(* CODESYS project Enums.export

Project tree, tasks and I/O mapping:
  Enums/
    data type DepositeProcessStage
    data type ERROR
    data type InficonMethodStage
    data type InficonMethodStatus
    data type InficonStage
    data type IPS_CONTROL_STAGE
    data type IPS_STATUS
    data type OWEN_TYPE
    data type PRESSURE_UNIT
    data type VACUUM_CAMERA_PROCESS_STAGE
    data type VACUUM_CAMERA_STATE
    TRM151/
      data type TRMAutomationCorrectionFreeEnds
      data type TRMInputNumberTrancitionValue
      data type TRMInputSensoreType
      data type TRMmanualChangeValue
      data type TRMNextStepTransactionLogic
      data type TRMObjectState
      data type TRMProgramPermit
      data type TRMRegulationMode
      data type TRMSetpointType
      data type TRMStartProgramSource
      data type TRMStartSignal
      data type TRMStepType
      data type TRMTimeFormat
      data type TRMTransactionConditionValue
      data type TRM_POOLING_STAGE
*)

// Enums/DepositeProcessStage
{attribute 'qualified_only'}
{attribute 'strict'}

TYPE DepositeProcessStage :
(
	WAIT_COMMAND 			:=0,  //Ожидание команды на старт
	INIT_DATA				:=10, //Инициализация уставок
	START_HEATER			:=11, //Включение источчника питания
	PREDEPOSITE_HEATING		:=15, //Этап нагрева по времени
	QARTZ_OPEN				:=20, //Открытие клапана кварцевого датчика
	QUARTZ_OPENED_DELAY		:=21, //Ожидание при открытом кварцевом датчике
	SOURCE_SHUTTER_OPEN		:=25, //Открытие залсонку источника напыления
	QARTZ_SENSORE_HEATING	:=30, //Прогрев кварцевого датчика для стабилизации показаний
	LIMIT_SPEED_DEPOSITE_1	:=35, //Напыление с заданной скоростью
	LIMIT_SPEED_DEPOSITE_2	:=36, //Наплыение с заданной скоростью
	STOP_DEPOSITE			:=40, //Остановка напыления
	ERROR					:=100 //Ошибка 
);
END_TYPE

// Enums/ERROR
{attribute 'qualified_only'}
//{attribute 'conditionalshow'}
//{attribute 'conditionalshow' := 'SomeText'}
//{attribute 'hide'}
TYPE ERROR : (NO_ERROR, TIME_OUT); END_TYPE

// Enums/InficonMethodStage
{attribute 'qualified_only'}
{attribute 'strict'}
TYPE InficonMethodStage :
(
	WAIT := 0,
	ADD_COMMAND:=1,
	ADD_LENGTH_TO_SENDBUFFER:=61,
	CALC_CRC:=70,
	ADD_CRC:=80,
	ADD_DATA_TO_SENDBUFFER:=90,
	EDGE_MESSAGECOMPLETE_FLAG:=91,
	WAIT_RESPONCE:=110,
	PARSE_RESPONCE:=120,
	CHECK_RESPONCE_STATUS:=121,
	COMPLETE:=130,
	ERROR:=140
);
END_TYPE

// Enums/InficonMethodStatus
{attribute 'qualified_only'}
{attribute 'strict'}
TYPE InficonMethodStatus :
(
	IDLE := 0,
	BUSY:=1,
	COMPLETE:=100,
	ERROR:=255
);
END_TYPE

// Enums/InficonStage
{attribute 'qualified_only'}
{attribute 'strict'}
TYPE InficonStage :
(
	WAIT := 0,
	STATUS_SENSORE:=10,
	GET_MATERIAL_FILTRED_RATE:=20,
	REMOTE_GENERAL_ACTION:=30,
	ERROR:=100
);
END_TYPE

// Enums/IPS_CONTROL_STAGE
{attribute 'qualified_only'}
{attribute 'strict'}
TYPE IPS_CONTROL_STAGE :
(
	WAIT := 0,
	START_PERMIT:=10,
	WAIT_PERMIT_ANSWER:=11,
	START:=20,
	WAIT_START_RESPONCE:=21,
	STOP:=30,
	WAIT_STOP_RESPONCE:=31,
	ERROR_RESET:=40,
	WAIT_ERROR_RESET_RESPONCE:=41,
	ERROR:=100
);
END_TYPE

// Enums/IPS_STATUS
{attribute 'qualified_only'}
{attribute 'strict'}
{attribute 'to_string'}
TYPE IPS_STATUS :
(
	PROCESS_RESET := 				769,	//Прошла инициализация устрйоства после включения питания
	START_PERMIT:=					10101,	//Разрешение выполнения ккоманды "Старт" выполнено без ошибок
	START_NO_ERROR:=				10001,	//Команда "старт" с  выполнена без ошибок
	START_KEYBORD_NO_ERROR:=		10201,	//Команда "старт" с клавитауры ввыполнена без ошибок
	START_CONTACT_NO_ERROR:=		10301, 	//Команда "Старт" с внешнего контакта выполнена без ошибок
	RUN_STEP_1:=					30101, 	//Выполняется команда "Старт" шаг 1
	RUN_STEP_2:=					30201,	//Выполняется команда "Старт" шаг 2
	RUN_STEP_3:=					30301,	//Выполняется команда "Старт" шаг 3
	RUN_STEP_4:=					30401,	//Выполняется команда "Старт" шаг 4
	RUN_STEP_5:=					30501,  //Выполняется команда "Старт" шаг 5
	RUN_STEP_6:=					30601,	//Выполняется команда "Старт" шаг 6
	RUN_STEP_7:=					30701,	//Выполняется команда "Старт" шаг 7
	RUN_STEP_7_1:=					30711, 	//Выполняется команда "Старт" шаг 7.1
	RUN_STEP_7_2:=					30721,	//Выполняется команда "Старт" шаг 7.2
	RUN_STEP_7_3:=					30731,	//Выполняется команда "Старт" шаг 7.3
	RUN_STEP_8:=					30801,	//Выполняется команда "Старт" шаг 8
	RUN_STEP_9:=					30901,	//Выполняется команда "Старт" шаг 9
	ERR_START_PERMIT:=				40101,	//Ошибка выполнения команда "Старт", нет разрешения старта
	ERR_START_ALARM:=				40201,	//Ошибка выполнения команды "Старт", активен сигнал авария
	ERR_START_POWER_SUPPLY:=		40301,	//Ошибка выполнения команды "Старт", напряжение истоника питная собственных нужд ниже нормы
	ERR_START_HIGHT_TEMPERATURE:=	40401,	//Ошибка выполнения команды "Старт" высокая температура воздуха
	ERR_START_HIGHT_TEMPERATURE_1:=	40501,	//Ошибка выполнения команды "Старт" высокая температура узлов устройства
	ERR_START_HIGHT_TEMPERATURE_2:= 40601,
	ERR_START_HIGHT_TEMPERATURE_3:= 40701,
	ERR_START_HIGHT_TEMPERATURE_4:= 41101,
	ERR_START_BLOCK_CONTACT:=		41001,	//Ошибка выполнения команды "Старт" контакт блокировки отключен
	ERR_START_ALREADY:=				41201,	//Ошибка выполнения команды "Старт" блок уже включен
	ERR_START_FILAMENT_CUT:=		41301,	//ошибка выполнения команды "Старт", обрыв нити накала
	ERR_START_GROUND_CUT:=			41501,	//Ошибка выполнения команды "Старт", обрыв заземления нагрузки
	ERR_START_DISPLAY_DISCONNECT:=	41601, 	//Ошибка выполнения команды "Старт", нет связи с дисплеем блока
	ERR_START_CONVERTER_MISSING:=	41701,	//Ошибка выполнения команды "Старт", нет подключенных преобразователей
	ERR_START_RMS_HOT:=				41801,	//Ошибка выполнения команды "Старт", датчик RMS горячий
	ERR_START_INTERNAL_CONNECT_1:=	41901,	//Ошибка выполнения команды "Старт", проблема со связью между узлами внутри блока
	ERR_START_INTERNAL_CONNECT_2:=	42001,
	ERR_START_INTERNAL_CONNECT_3:=	42101,
	ERR_START_STOP_DELAY:=			42201,	//Ошибка выполнения команды "Старт", пауза после выключения меньше 3 секунд
	ERR_START_RUN_CONVERTER_ERR:=	42301,	//Ошибка выполнения команды "Старт", проблемы с пуском преобразователя
	ERR_START_ADC_DISCONNECT:=		42601,	//Ошибка выполнения команды "Старт", нет связи с АЦП контроля выходного напрядения устройства
	STOP_NO_ERROR:=					10002,	//Команда "Стоп" выполнена
	STOP_KEYBORD_NO_ERROR:=			10102,	//Команда "Стоп" выполнена по нажатию кнопки "Стоп"
	STOP_CONTACT_NO_ERROR:=			10202,	//Команда "Стоп" выполнена по вненему контакту
	STOP_AFTER_SMOOTH_SHUTDOWN_FILAMENT:=	10501, //Команда "Стоп" выполнена после плавного отключения накала
	STOP_ANOD_CHANELL:=				10602,	//Команда "Стоп" выполнена для канала анода
	EMG_STOP_ALARM:=				40202,	//Аварийный "Стоп по сигналу "Авария"
	EMG_STOP_POWER_SUPPLY:=			40302,	//Аварийный "Стоп", напряжение источника питания собственных нужд ниже нормы
	EMG_STOP_HOT_AIR:=				40402,	//Авариынй "Стоп", горячий воздух
	EMG_STOP_OVERHEAT_1:=			40502,	//Аварийный "Стоп", перегрев узлоа
	EMG_STOP_OVERHEAT_2:=			40602,
	EMG_STOP_OVERHEAT_3:=			40702,
	EMG_STOP_OVERHEAT_4:=			41102,
	EMG_STOP_WATCHDOG:=				40802,	//Аварийный "Стоп" сработал сторожевой таймер
	EMG_STOP_INTERLOCK:=			41002,	//Аварийный "Стоп", сработал внешний блокировочный контакт
	EMG_STOP_FILAMENT_ALARM:=		41302,	//Аварийный "Стоп", авария накала
	EMG_STOP_INTERNAL_SYNC_MISSING:=41402,	//Аварийный "Стоп", потеря внетренней синхронизации между узлами устройства
	EMG_STOP_GROUND_CUT:=			41502,	//Аварийный "Стоп", обрыв заземления нагрузки
	EMG_STOP_INTERNAL_CONNECT_1:=	41602,	//аварийный "Стоп", ошибка связи между узлами устройства
	EMG_STOP_INTERNAL_CONNECT_2:=	41902,
	EMG_STOP_INTERNAL_CONNECT_3:=	42002,
	EMG_STOP_INTERNAL_CONNECT_4:=	42102,
	EMG_STOP_RMS_OVERLOAD:=			41802,	//Аварийный "Стоп", большой ток RMS
	EMG_STOP_CONVERTER_EMG_RELOAD:=	42202,	//Аварийный "Стоп", аварийный перезапуцск преобразователя
	EMG_STOP_LOW_VOLTAGE:=			42302,	//Аварийный "Стоп", напряжение нагрузки ниже нормы
	EMG_STOP_ADC_DISCONNECT:=		42602, 	//Аварийный "Стоп", нет связи с АЦП контроля выходного напряжения устройства
	RESET_ERROR_DONE:=				10003, 	//Команда "Сброс ошибок" выполнена
	RESET_ERROR_AFTER_STOP:=		10103, 	//Команда "Сброс ошибок" выполнена по нажатию кнопки "Стоп"
	RESET_ERROR_FAIl:=				40003	//Команда "Сброс ошибок" не выполнена, устройство в режиме "Старт"
	
);
END_TYPE

// Enums/OWEN_TYPE
{attribute 'qualified_only'}
{attribute 'strict'}
TYPE OWEN_TYPE :
(
	INTEGER 	:= 0,
	FLOAT		:=1,
	OTHER		:=2
);
END_TYPE

// Enums/PRESSURE_UNIT
{attribute 'qualified_only'}
{attribute 'strict'}
TYPE PRESSURE_UNIT :
(
	mBar := 0,
	Pascal:=1,
	Torr:=2
);
END_TYPE

// Enums/VACUUM_CAMERA_PROCESS_STAGE
{attribute 'qualified_only'}
{attribute 'strict'}
TYPE VACUUM_CAMERA_PROCESS_STAGE :
(
	WAIT := 0, //Ожидание
	START_VACUUM_PROCESS:=10,//Старт процессса откачки вакуумной камеры
	START_VACUUM_PROCESS_CHECK_FVP_SELECT:=11,//Проверка ФВП на флаг работоспособности
	START_VACUUM_PROCESS_CHECKING_FVP:=12,//Проверка ФВН на рпботоспособнтсть
	START_VACUUM_PROCESS_FORVACUUMING_PROCESS:=13,//Процесс форвакуумной откачка
	START_VACUUM_PROCESS_TMP_FORVACUUMING_PROCESS:=14,//Процесс откачки через форвакуумный насосо и ТМН
	START_VACUUM_PROCESS_TMP_START:=15,//Запуск ТМН
	START_VACUUM_PROCESS_COMPLETE_WAIT:=16,//Ожидание завершения процессаы
	START_REVACUUM_PROCESS:=20,//Старт процесса повтороной откачки вакуумнйо камеры
	
	
	START_DEVACUUM_PROCESS:=30,//Старт процесса напуска атмосферы в вакуумную камеру
	START_DEVACUUM_STOP_TMP:=31,//Старт полного цикла остановки
	START_DEVACUUM_STOP_FVP:=32,
	START_DEVACUUM_OPEN_CAM:=33,

	
	
	
	
	STOP_VACUUM_PROCESS:=40,//остановка работы вакуумной камеры
	STOP_ANY_PROCESS:=50, //Стадия остановки любого процесса
	ERROR:=1000//Ошибка в работе алгоритма
);
END_TYPE

// Enums/VACUUM_CAMERA_STATE
{attribute 'qualified_only'}
{attribute 'strict'}
TYPE VACUUM_CAMERA_STATE :
(
	CAMERA_NOT_VACUUM := 0,	//Камера находится не под вакуумом
	CAMERA_VACUUM:=10 		//Камера находится по двакуумом
	
);
END_TYPE

// Enums/TRM151/TRMAutomationCorrectionFreeEnds
{attribute 'qualified_only'}
{attribute 'strict'}
TYPE TRMAutomationCorrectionFreeEnds :
(
	OFF := 1,
	ON	:=2
);
END_TYPE

// Enums/TRM151/TRMInputNumberTrancitionValue
{attribute 'qualified_only'}
{attribute 'strict'}
(*
Номер входа, величина с которого должна достичь значение уставки
*)
TYPE TRMInputNumberTrancitionValue :
(
	OFF := 0,
	Input_1:=1,
	Input_2:=2
);
END_TYPE

// Enums/TRM151/TRMInputSensoreType
{attribute 'qualified_only'}
{attribute 'strict'}
TYPE TRMInputSensoreType :
(
	DISABLE := 0,
	TSM100M :=1,
	TSM50M:=2,
	TSP100P_1_385:=3,
	TSP100P_1_391:=4,
	THK_L:=5,
	THA_K:=6,
	Sensore50vM:=7,
	TSP50_1_385:=8,
	TSP50_1_391:=9,
	Sensore_4_20ma:=11,
	Sensore_0_20ma:=12,
	Sensore_0_5ma:=13,
	Sensore_0_1V:=14,
	TPR_B:=17,
	TPP_S:=18,
	TPP_R:=19,
	TNN_N:=20,
	TJK_J:=21,
	TVR_A_1:=22,
	TVR_A_2:=23,
	TVR_A_3:=24,
	TMK_T:=25
	
);
END_TYPE

// Enums/TRM151/TRMmanualChangeValue
{attribute 'qualified_only'}
{attribute 'strict'}
TYPE TRMmanualChangeValue :
(
	Enable := 0,
	Disable:=1
);
END_TYPE

// Enums/TRM151/TRMNextStepTransactionLogic
{attribute 'qualified_only'}
{attribute 'strict'}
(*Логика перехода на следующий шаг*)
TYPE TRMNextStepTransactionLogic :
(
	GetLimitValue := 1, //По достижению порогового ззначения
	GetTime:=2,			//по времения
	GetLimitValueAndtime:=3,//По достижению порогового значени и времени
	GetLimitValueOrtime:=4
);
END_TYPE

// Enums/TRM151/TRMObjectState
{attribute 'qualified_only'}
{attribute 'strict'}
TYPE TRMObjectState :
(
	Stop := 0,								//Останов
	Work:=1,								//Работа
	WaitWorkCondition:=2,					//Ожидание условий запуска
	Pause:=3,								//пауза
	WaitWorkConditionAfterPowerFailure:=4,	//Ожидание условй запуска после пропадания питания
	GraphicSetMode:=5,						//Режим задания графиков
	ChooseProgrammAndStep:=6,				//Выбор программы и шага
	StopAfterComplite:=7,					//Остановка после выполнения программы
	FailureWithAlarm:=8,					//авария с сигнализацией
	FailureWithoutAlarm:=9					//Авария без сигнализации
);
END_TYPE

// Enums/TRM151/TRMProgramPermit
{attribute 'qualified_only'}
{attribute 'strict'}
(*Разрешение на заупск программы*)
TYPE TRMProgramPermit :
(
	Accept := 1,
	Decline:=2
);
END_TYPE

// Enums/TRM151/TRMRegulationMode
{attribute 'qualified_only'}
{attribute 'strict'}
TYPE TRMRegulationMode :
(
	TwoPosition := 0,
	PIDReg		:=1
);
END_TYPE

// Enums/TRM151/TRMSetpointType
{attribute 'qualified_only'}
{attribute 'strict'}
TYPE TRMSetpointType :
(
	Temperature := 0,
	Power:=1
);
END_TYPE

// Enums/TRM151/TRMStartProgramSource
{attribute 'qualified_only'}
{attribute 'strict'}
TYPE TRMStartProgramSource :
(
	SelfLogic := 1,
	NetCommand:=2
);
END_TYPE

// Enums/TRM151/TRMStartSignal
{attribute 'qualified_only'}
{attribute 'strict'}
(*сигналы на старт*)
TYPE TRMStartSignal :
(
	STOP 	:= 0,
	RUN		:= 1,
	PAUSE	:= 2
);
END_TYPE

// Enums/TRM151/TRMStepType
{attribute 'qualified_only'}
{attribute 'strict'}
TYPE TRMStepType :
(
	BasicStep := 1,
	TransitionStep:=2,
	ProgramEnd:=3
);
END_TYPE

// Enums/TRM151/TRMTimeFormat
{attribute 'qualified_only'}
{attribute 'strict'}
TYPE TRMTimeFormat :
(
	HoursMinutes := 1,
	MinutesSeconds:=2
);
END_TYPE

// Enums/TRM151/TRMTransactionConditionValue
{attribute 'qualified_only'}
{attribute 'strict'}
(*Условия при переходе по пороговому значению*)
TYPE TRMTransactionConditionValue :
(
	LessThenLimitValue := 1, //переход если стало меньше порога
	MoreThenLimitValue :=2	//Переход елси стало больше порога
);
END_TYPE

// Enums/TRM151/TRM_POOLING_STAGE
{attribute 'qualified_only'}
{attribute 'strict'}
(*
	Список стадий обмена сообщениями с ТРМ
*)
TYPE TRM_POOLING_STAGE :
(
	WAIT := 0, 						//Ожидание
	GET_ACTION:=1, 					//Получение данных из очереди
	ChanellTRM_SAVE:=10, 			//Сохранение данных канала
	InputTRM_SAVE:=20,				//Сохранение данных входных значений
	OutputTRM_SAVE:=30,				//Сохранение данных выходных значений
	ProgramOfTechonologTRM_SAVE:=40,//Сохранение данных прогррамы технолога
	ProgramOfTechonologTRM_SETPOINT_SAVE:=41,//Сохранение данных прогррамы технолога
	OperatingTRM_SAVE:=50,			//Сохранение оперативных параметров
	OperatingTRM_LOAD:=60,			//Загрузка оперативных параметров
	OperatingTRM_STARTSTOP:=70,		//Сохранение параметров старт стоп
	ERROR:=80						//
);
END_TYPE
